// TwinCAT 3 PLC project ProxyPLC
// ProgramVersion: 3.1.4026.22
// libraries:
//   Tc2_Standard, * (Beckhoff Automation GmbH)
//   Tc2_System, * (Beckhoff Automation GmbH)
// project tree:
//   POUs/ FB_DoWork.TcPOU, MAIN.TcPOU
// (motion and I/O tree: see PLC project plc1)
// real-time tasks:
//   TASK Plc1Task: cycle T#10ms, priority 20, ADS port 350
//   TASK Plc2Task: cycle T#10ms, priority 21, ADS port 351

// ---- POUs/FB_DoWork.TcPOU
FUNCTION_BLOCK FB_DoWork EXTENDS TcBaseModuleRegistered
VAR_INPUT
END_VAR
VAR_OUTPUT
END_VAR
VAR
END_VAR

{attribute 'TcTypeSystem'}
{attribute 'c++_compatible'}
{attribute 'minimal_input_size' := '4'}
{attribute 'pack_mode' := '4'}
{warning 'Add method implementation '}
METHOD GetClassId : Global.HRESULT
VAR_INPUT
	classId	: REFERENCE TO Global.CLSID;
END_VAR
END_METHOD

{attribute 'TcTypeSystem'}
{attribute 'c++_compatible'}
{attribute 'minimal_input_size' := '4'}
{attribute 'pack_mode' := '4'}
{warning 'Add method implementation '}
METHOD TcAddRef : UDINT
END_METHOD

{attribute 'TcTypeSystem'}
{attribute 'c++_compatible'}
{attribute 'minimal_input_size' := '4'}
{attribute 'pack_mode' := '4'}
{warning 'Add method implementation '}
METHOD TcGetObjectId : Global.HRESULT
VAR_INPUT
	objId	: REFERENCE TO Global.OTCID;
END_VAR
END_METHOD

{attribute 'TcTypeSystem'}
{attribute 'c++_compatible'}
{attribute 'minimal_input_size' := '4'}
{attribute 'pack_mode' := '4'}
{warning 'Add method implementation '}
METHOD TcGetObjectName : Global.HRESULT
VAR_INPUT
	objName	: POINTER TO SINT;
	nameLen	: UDINT;
END_VAR
END_METHOD

{attribute 'TcTypeSystem'}
{attribute 'c++_compatible'}
{attribute 'minimal_input_size' := '4'}
{attribute 'pack_mode' := '4'}
{warning 'Add method implementation '}
METHOD TcGetObjPara : Global.HRESULT
VAR_INPUT
	pid	: Global.PTCID;
	nData	: REFERENCE TO UDINT;
	pData	: REFERENCE TO Global.PVOID;
	pgp	: Global.PTCGP := 0;
END_VAR
END_METHOD

{attribute 'TcTypeSystem'}
{attribute 'c++_compatible'}
{attribute 'minimal_input_size' := '4'}
{attribute 'pack_mode' := '4'}
{warning 'Add method implementation '}
METHOD TcGetObjState : Global.HRESULT
VAR_INPUT
	pState	: POINTER TO Global.TCOM_STATE;
END_VAR
END_METHOD

{attribute 'TcTypeSystem'}
{attribute 'c++_compatible'}
{attribute 'minimal_input_size' := '4'}
{attribute 'pack_mode' := '4'}
{warning 'Add method implementation '}
METHOD TcGetParentObjId : Global.HRESULT
VAR_INPUT
	objId	: REFERENCE TO Global.OTCID;
END_VAR
END_METHOD

{attribute 'TcTypeSystem'}
{attribute 'c++_compatible'}
{attribute 'minimal_input_size' := '4'}
{attribute 'pack_mode' := '4'}
{warning 'Add method implementation '}
METHOD TcQueryInterface : Global.HRESULT
VAR_INPUT
	iid	: REFERENCE TO Global.IID;
	pipItf	: POINTER TO Global.PVOID;
END_VAR
END_METHOD

{attribute 'TcTypeSystem'}
{attribute 'c++_compatible'}
{attribute 'minimal_input_size' := '4'}
{attribute 'pack_mode' := '4'}
{warning 'Add method implementation '}
METHOD TcRelease : UDINT
END_METHOD

{attribute 'TcTypeSystem'}
{attribute 'c++_compatible'}
{attribute 'minimal_input_size' := '4'}
{attribute 'pack_mode' := '4'}
{warning 'Add method implementation '}
METHOD TcSetObjectId : Global.HRESULT
VAR_INPUT
	objId	: Global.OTCID;
END_VAR
END_METHOD

{attribute 'TcTypeSystem'}
{attribute 'c++_compatible'}
{attribute 'minimal_input_size' := '4'}
{attribute 'pack_mode' := '4'}
{warning 'Add method implementation '}
METHOD TcSetObjectName : Global.HRESULT
VAR_INPUT
	objName	: POINTER TO SINT;
END_VAR
END_METHOD

{attribute 'TcTypeSystem'}
{attribute 'c++_compatible'}
{attribute 'minimal_input_size' := '4'}
{attribute 'pack_mode' := '4'}
{warning 'Add method implementation '}
METHOD TcSetObjPara : Global.HRESULT
VAR_INPUT
	pid	: Global.PTCID;
	nData	: UDINT;
	pData	: Global.PVOID;
	pgp	: Global.PTCGP := 0;
END_VAR
END_METHOD

{attribute 'TcTypeSystem'}
{attribute 'c++_compatible'}
{attribute 'minimal_input_size' := '4'}
{attribute 'pack_mode' := '4'}
{warning 'Add method implementation '}
METHOD TcSetObjState : Global.HRESULT
VAR_INPUT
	state	: Global.TCOM_STATE;
	ipSrv	: Global.ITComObjectServer;
	pInitData	: POINTER TO Global.TComInitDataHdr;
END_VAR
END_METHOD

{attribute 'TcTypeSystem'}
{attribute 'c++_compatible'}
{attribute 'minimal_input_size' := '4'}
{attribute 'pack_mode' := '4'}
{warning 'Add method implementation '}
METHOD TcSetParentObjId : Global.HRESULT
VAR_INPUT
	objId	: Global.OTCID;
END_VAR
END_METHOD

END_FUNCTION_BLOCK

// ---- POUs/MAIN.TcPOU
PROGRAM MAIN
VAR
END_VAR

END_PROGRAM
